PROGRAM LinkUI
VAR
	bTemp		:BOOL;
END_VAR

GVL_SignalHanlding.fbPauseUI();
GVL_SignalHanlding.fbPauseUI.SignalEnable(bSignalLocalEnable:= TRUE);
GVL_SignalHanlding.fbPauseUI.SetOutput();
//bTemp := GVL_SignalHanlding.fbPauseUI.bSignalOutput;

END_PROGRAM

(* stored: Version 1.1.0.1, ProductVersion 3.1.4022.16
   POU LinkUI: Id {1a1c3c5e-22cb-45b4-b980-f09563072448}, SpecialFunc None *)
